// TIA Portal project "Project21" (V19)

(* hardware
DEVICE "S7-1200 station_1"  S7-1200 Station
   slot 0: "Rack_0"  S7-1200 Rack  Rack  V1.0
   slot 1: "PLC_1"  CPU 1215C DC/DC/DC  6ES7 215-1AG40-0XB0  V4.5
*)

// ===== PLC "PLC_1"  CPU 1215C DC/DC/DC =====

VAR_GLOBAL   // PLC tag table "Default tag table"
   "Encendido" AT %M0.0 : Bool;
   "ManAuto" AT %M0.1 : Bool;
   "System_Byte" AT %MB1 : Byte;
   "FirstScan" AT %M1.0 : Bool;
   "DiagStatusUpdate" AT %M1.1 : Bool;
   "AlwaysTRUE" AT %M1.2 : Bool;
   "AlwaysFALSE" AT %M1.3 : Bool;
END_VAR

DATA_BLOCK "DB_SimVent"   // DB1
{ S7_Optimized_Access := 'TRUE' }
VERSION : 0.1
// stored: InstanceOfName FB_Simulacion
"FB_Simulacion"
BEGIN
END_DATA_BLOCK

DATA_BLOCK "DB_HMIET"   // DB2
{ S7_Optimized_Access := 'FALSE' }
VERSION : 0.1
   VAR
      TEMPERATURA_SP : Real := 22.0;
      HUMEDAD_SP : Real := 60.0;
      PRESION_SP : Real := 1016.0;
      VENT_VEL_OUT : Real := 799.0;
      BOMBA_VEL_OUT : Real := 1434.0;
      CTRL_DESHUM : Int;
      CTRL_ENFRIAM_CALEF : Int;
      SPTEMP : Real;
      SPHUM : Real;
      SPPRE : Real;
      TEMPERATURA_HMI : Int;
      HUMEDAD_HMI : Int;
      PRESION_HMI : Int;
      ENFRIAMIENTO_HMI : Bool;
      CALEFACCION_HMI : Bool;
      DESHUM_HMI : Bool;
      AutoMan : Bool;
      SPTEMP_HMI : Real;
      SPHUM_HMI : Real;
      SPPRE_HMI : Real;
   END_VAR
BEGIN
END_DATA_BLOCK

DATA_BLOCK "DM_SimTemp"   // DB3
{ S7_Optimized_Access := 'TRUE' }
VERSION : 0.1
// stored: InstanceOfName FB_Simulacion
"FB_Simulacion"
BEGIN
   PVIn := 19.0;
END_DATA_BLOCK

DATA_BLOCK "DB_SimPresion"   // DB4
{ S7_Optimized_Access := 'TRUE' }
VERSION : 0.1
// stored: InstanceOfName FB_Simulacion
"FB_Simulacion"
BEGIN
   PVIn := 1000.0;
END_DATA_BLOCK

DATA_BLOCK "DB_SimHumedad"   // DB5
{ S7_Optimized_Access := 'TRUE' }
VERSION : 0.1
// stored: InstanceOfName FB_Simulacion
"FB_Simulacion"
BEGIN
   PVIn := 50.0;
END_DATA_BLOCK

DATA_BLOCK "DB_SimBomba"   // DB6
{ S7_Optimized_Access := 'TRUE' }
VERSION : 0.1
// stored: InstanceOfName FB_Simulacion
"FB_Simulacion"
BEGIN
END_DATA_BLOCK

DATA_BLOCK "DB_HMIOUT"   // DB7
{ S7_Optimized_Access := 'FALSE' }
VERSION : 0.1
   VAR
      PRESION_OUT : Real;
      HUMEDAD_OUT : Real;
      TEMPERATURA_OUT : Real;
   END_VAR
BEGIN
END_DATA_BLOCK

FUNCTION_BLOCK "FB_Simulacion"   // FB2, LAD
{ S7_Optimized_Access := 'TRUE' }
VERSION : 0.1
   VAR_INPUT
      Encendido : Bool;
      ManAuto : Bool;
      MS : Real;
      MI : Real;
      PVIn : Real;
      SP : Real;
   END_VAR
   VAR_OUTPUT
      PVOut : Real;
      Ctrl : Int;
   END_VAR
   VAR
      TON_Simulacion : TON_TIME;
      ResetTimerSim : Bool;
      Sim1 : Bool;
      Sim2 : Bool;
      Sim3 : Bool;
      Timer_Ajuste : TON_TIME;
      ResetTimerAjuste : Bool;
      Estado : Int;
      MSSP : Real;
      MISP : Real;
      FinSim1 : Bool;
      FinSim2 : Bool;
      EnclavEstado : Bool;
      Timer_ManAuto : TON_TIME;
   END_VAR
   VAR_TEMP   // added for the SCL form of the ladder/FBD networks
      _w1 : Bool;
      _w2 : Bool;
   END_VAR
BEGIN

REGION Network 1
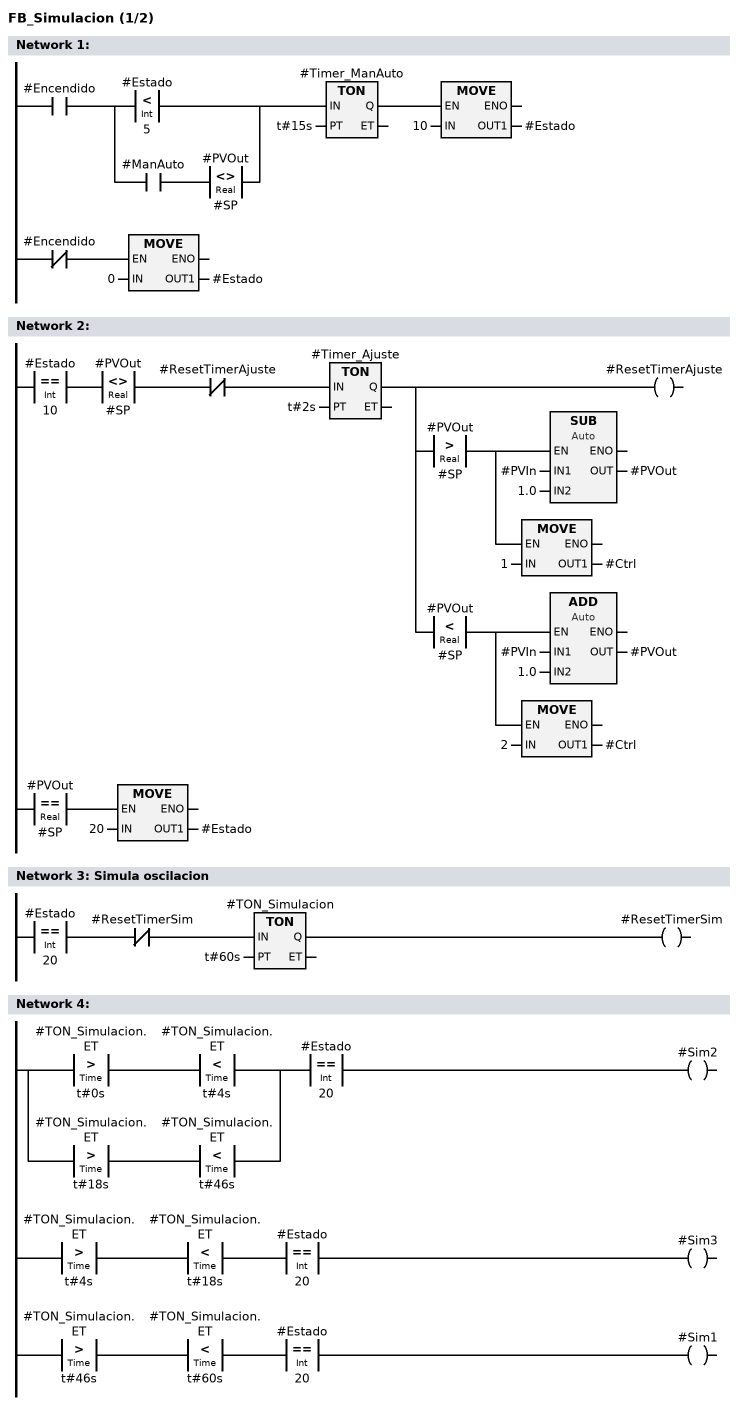
   #Timer_ManAuto(IN := #Encendido AND ((#Estado < 5) OR (#ManAuto AND (#PVOut <> #SP))), PT := t#15s);   // TON
   IF #Timer_ManAuto.Q THEN #Estado := 10; END_IF;
   IF NOT #Encendido THEN #Estado := 0; END_IF;
END_REGION

REGION Network 2
   #Timer_Ajuste(IN := (#Estado = 10) AND (#PVOut <> #SP) AND NOT #ResetTimerAjuste, PT := t#2s);   // TON
   #ResetTimerAjuste := #Timer_Ajuste.Q;
   #_w1 := #Timer_Ajuste.Q AND (#PVOut > #SP);
   IF #_w1 THEN
       #PVOut := #PVIn - 1.0;
       #Ctrl := 1;
   END_IF;
   #_w2 := #Timer_Ajuste.Q AND (#PVOut < #SP);
   IF #_w2 THEN
       #PVOut := #PVIn + 1.0;
       #Ctrl := 2;
   END_IF;
   IF #PVOut = #SP THEN #Estado := 20; END_IF;
END_REGION

REGION Network 3: Simula oscilacion
   #TON_Simulacion(IN := (#Estado = 20) AND NOT #ResetTimerSim, PT := t#60s);   // TON
   #ResetTimerSim := #TON_Simulacion.Q;
END_REGION

REGION Network 4
   RUNG wire#powerrail
      { S7_Templates := "SrcType := Time" } GT_Contact(in1 := #TON_Simulacion.ET, in2 := t#0s)
      { S7_Templates := "SrcType := Time" } LT_Contact(in1 := #TON_Simulacion.ET, in2 := t#4s)
      wire#w1
      { S7_Templates := "SrcType := Int" } EQ_Contact(in1 := #Estado, in2 := 20)
      Coil( #Sim2 )
   END_RUNG
   RUNG wire#powerrail
      { S7_Templates := "SrcType := Time" } GT_Contact(in1 := #TON_Simulacion.ET, in2 := t#18s)
      { S7_Templates := "SrcType := Time" } LT_Contact(in1 := #TON_Simulacion.ET, in2 := t#46s)
   END_RUNG wire#w1
   RUNG wire#powerrail
      { S7_Templates := "SrcType := Time" } GT_Contact(in1 := #TON_Simulacion.ET, in2 := t#4s)
      { S7_Templates := "SrcType := Time" } LT_Contact(in1 := #TON_Simulacion.ET, in2 := t#18s)
      { S7_Templates := "SrcType := Int" } EQ_Contact(in1 := #Estado, in2 := 20)
      Coil( #Sim3 )
   END_RUNG
   RUNG wire#powerrail
      { S7_Templates := "SrcType := Time" } GT_Contact(in1 := #TON_Simulacion.ET, in2 := t#46s)
      { S7_Templates := "SrcType := Time" } LT_Contact(in1 := #TON_Simulacion.ET, in2 := t#60s)
      { S7_Templates := "SrcType := Int" } EQ_Contact(in1 := #Estado, in2 := 20)
      Coil( #Sim1 )
   END_RUNG
   // the same network as SCL:
   #Sim2 := (((#TON_Simulacion.ET > t#0s) AND (#TON_Simulacion.ET < t#4s)) OR ((#TON_Simulacion.ET > t#18s) AND (#TON_Simulacion.ET < t#46s))) AND (#Estado = 20);
   #Sim3 := (#TON_Simulacion.ET > t#4s) AND (#TON_Simulacion.ET < t#18s) AND (#Estado = 20);
   #Sim1 := (#TON_Simulacion.ET > t#46s) AND (#TON_Simulacion.ET < t#60s) AND (#Estado = 20);
END_REGION

REGION Network 5
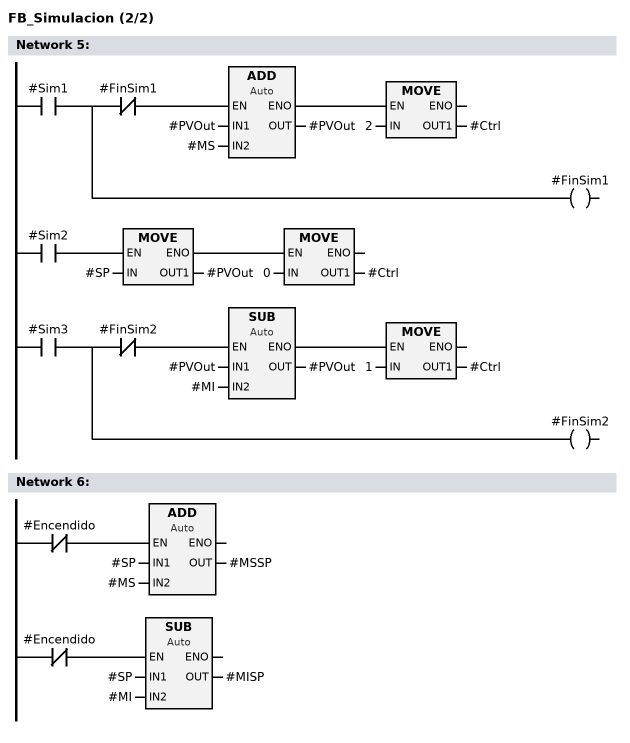
   RUNG wire#powerrail
      Contact( #Sim1 )
      wire#w1
      I_Contact( #FinSim1 )
      Add(in1 := #PVOut, in2 := #MS, out => #PVOut)
      Move(in := 2, out1 => #Ctrl)
   END_RUNG
   RUNG wire#w1
      Coil( #FinSim1 )
   END_RUNG
   RUNG wire#powerrail
      Contact( #Sim2 )
      Move(in := #SP, out1 => #PVOut)
      Move(in := 0, out1 => #Ctrl)
   END_RUNG
   RUNG wire#powerrail
      Contact( #Sim3 )
      wire#w2
      I_Contact( #FinSim2 )
      Sub(in1 := #PVOut, in2 := #MI, out => #PVOut)
      Move(in := 1, out1 => #Ctrl)
   END_RUNG
   RUNG wire#w2
      Coil( #FinSim2 )
   END_RUNG
   // the same network as SCL:
   IF #Sim1 AND NOT #FinSim1 THEN
       #PVOut := #PVOut + #MS;
       #Ctrl := 2;
   END_IF;
   #FinSim1 := #Sim1;
   IF #Sim2 THEN
       #PVOut := #SP;
       #Ctrl := 0;
   END_IF;
   IF #Sim3 AND NOT #FinSim2 THEN
       #PVOut := #PVOut - #MI;
       #Ctrl := 1;
   END_IF;
   #FinSim2 := #Sim3;
END_REGION

REGION Network 6
   RUNG wire#powerrail
      I_Contact( #Encendido )
      Add(in1 := #SP, in2 := #MS, out => #MSSP)
   END_RUNG
   RUNG wire#powerrail
      I_Contact( #Encendido )
      Sub(in1 := #SP, in2 := #MI, out => #MISP)
   END_RUNG
   // the same network as SCL:
   IF NOT #Encendido THEN
       #MSSP := #SP + #MS;
       #MISP := #SP - #MI;
   END_IF;
END_REGION
END_FUNCTION_BLOCK

FUNCTION "FC_ConversionEscalado" : Void   // FC1, LAD
{ S7_Optimized_Access := 'TRUE' }
VERSION : 0.1
   VAR_INPUT
      EntradaInt : Int;
      MinNorm : Int;
      MaxNorm : Int;
      MinReal : Real;
      MaxReal : Real;
   END_VAR
   VAR_OUTPUT
      SalidaReal : Real;
   END_VAR
   VAR_TEMP
      IntReal : Real;
      RealNorm : Real;
   END_VAR
BEGIN

REGION Network 1
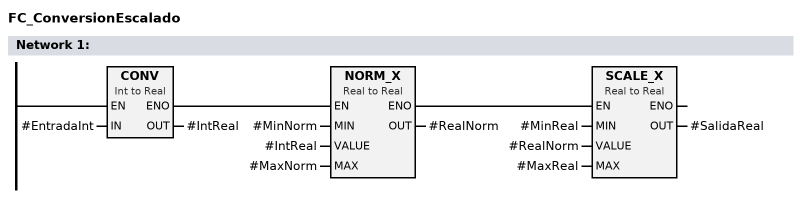
   RUNG wire#powerrail
      { S7_Templates := "[SrcType := Int, DestType := Real]" } Convert(in := #EntradaInt, out => #IntReal)
      { S7_Templates := "[SrcType := Real, DestType := Real]" } Normalize(min := #MinNorm, value := #IntReal, max := #MaxNorm, out => #RealNorm)
      { S7_Templates := "[SrcType := Real, DestType := Real]" } Scale(min := #MinReal, value := #RealNorm, max := #MaxReal, out => #SalidaReal)
   END_RUNG
   // the same network as SCL:
   #IntReal := INT_TO_REAL(#EntradaInt);
   #RealNorm := NORM_X(MIN := #MinNorm, VALUE := #IntReal, MAX := #MaxNorm);
   #SalidaReal := SCALE_X(MIN := #MinReal, VALUE := #RealNorm, MAX := #MaxReal);
END_REGION
END_FUNCTION

ORGANIZATION_BLOCK "Main"   // OB1, LAD, ProgramCycle
TITLE = "Main Program Sweep (Cycle)"
{ S7_Optimized_Access := 'TRUE' }
VERSION : 0.1
   VAR_INPUT
      Initial_Call : Bool;   // Initial call of this OB
      Remanence : Bool;   // =True, if remanent data are available
   END_VAR
   VAR_TEMP
      SPTEMP_ESC : Real;
      SPHUM_ESC : Real;
      SPPRE_ESC : Real;
   END_VAR
BEGIN

REGION Network 1
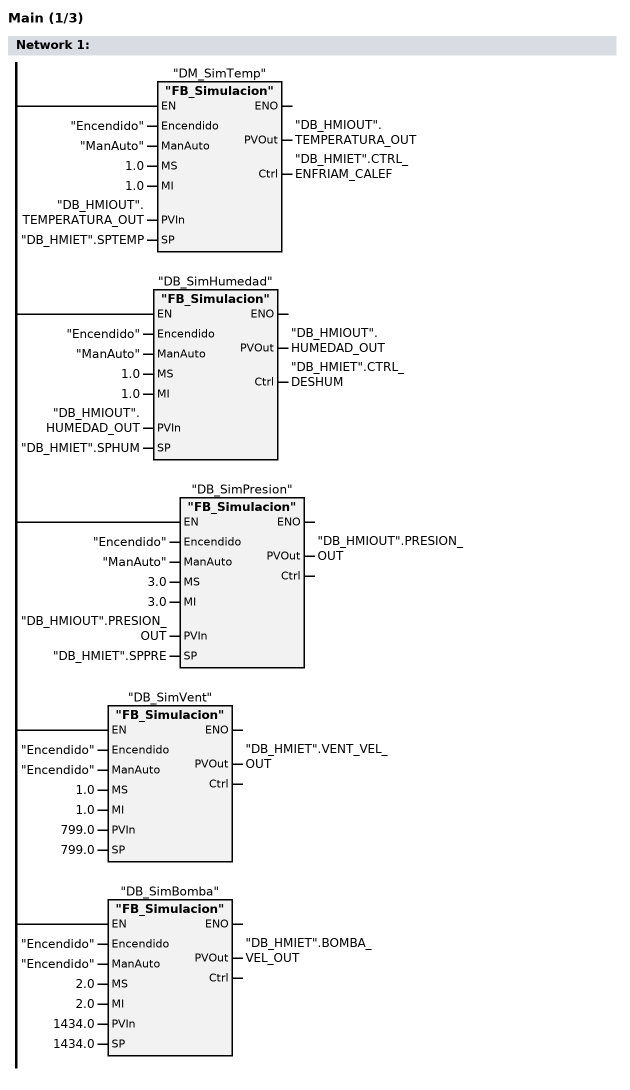
   RUNG wire#powerrail
      "DM_SimTemp"(Encendido := "Encendido", ManAuto := "ManAuto", MS := 1.0, MI := 1.0, PVIn := "DB_HMIOUT".TEMPERATURA_OUT, SP := "DB_HMIET".SPTEMP, PVOut => "DB_HMIOUT".TEMPERATURA_OUT, Ctrl => "DB_HMIET".CTRL_ENFRIAM_CALEF)
   END_RUNG
   RUNG wire#powerrail
      "DB_SimHumedad"(Encendido := "Encendido", ManAuto := "ManAuto", MS := 1.0, MI := 1.0, PVIn := "DB_HMIOUT".HUMEDAD_OUT, SP := "DB_HMIET".SPHUM, PVOut => "DB_HMIOUT".HUMEDAD_OUT, Ctrl => "DB_HMIET".CTRL_DESHUM)
   END_RUNG
   RUNG wire#powerrail
      "DB_SimPresion"(Encendido := "Encendido", ManAuto := "ManAuto", MS := 3.0, MI := 3.0, PVIn := "DB_HMIOUT".PRESION_OUT, SP := "DB_HMIET".SPPRE, PVOut => "DB_HMIOUT".PRESION_OUT, Ctrl =>)
   END_RUNG
   RUNG wire#powerrail
      "DB_SimVent"(Encendido := "Encendido", ManAuto := "Encendido", MS := 1.0, MI := 1.0, PVIn := 799.0, SP := 799.0, PVOut => "DB_HMIET".VENT_VEL_OUT, Ctrl =>)
   END_RUNG
   RUNG wire#powerrail
      "DB_SimBomba"(Encendido := "Encendido", ManAuto := "Encendido", MS := 2.0, MI := 2.0, PVIn := 1434.0, SP := 1434.0, PVOut => "DB_HMIET".BOMBA_VEL_OUT, Ctrl =>)
   END_RUNG
   // the same network as SCL:
   "DM_SimTemp"(Encendido := "Encendido",   // "FB_Simulacion"
                ManAuto := "ManAuto",
                MS := 1.0,
                MI := 1.0,
                PVIn := "DB_HMIOUT".TEMPERATURA_OUT,
                SP := "DB_HMIET".SPTEMP,
                PVOut => "DB_HMIOUT".TEMPERATURA_OUT,
                Ctrl => "DB_HMIET".CTRL_ENFRIAM_CALEF);
   "DB_SimHumedad"(Encendido := "Encendido",   // "FB_Simulacion"
                   ManAuto := "ManAuto",
                   MS := 1.0,
                   MI := 1.0,
                   PVIn := "DB_HMIOUT".HUMEDAD_OUT,
                   SP := "DB_HMIET".SPHUM,
                   PVOut => "DB_HMIOUT".HUMEDAD_OUT,
                   Ctrl => "DB_HMIET".CTRL_DESHUM);
   "DB_SimPresion"(Encendido := "Encendido",   // "FB_Simulacion"
                   ManAuto := "ManAuto",
                   MS := 3.0,
                   MI := 3.0,
                   PVIn := "DB_HMIOUT".PRESION_OUT,
                   SP := "DB_HMIET".SPPRE,
                   PVOut => "DB_HMIOUT".PRESION_OUT);
   "DB_SimVent"(Encendido := "Encendido",   // "FB_Simulacion"
                ManAuto := "Encendido",
                MS := 1.0,
                MI := 1.0,
                PVIn := 799.0,
                SP := 799.0,
                PVOut => "DB_HMIET".VENT_VEL_OUT);
   "DB_SimBomba"(Encendido := "Encendido",   // "FB_Simulacion"
                 ManAuto := "Encendido",
                 MS := 2.0,
                 MI := 2.0,
                 PVIn := 1434.0,
                 SP := 1434.0,
                 PVOut => "DB_HMIET".BOMBA_VEL_OUT);
END_REGION

REGION Network 2
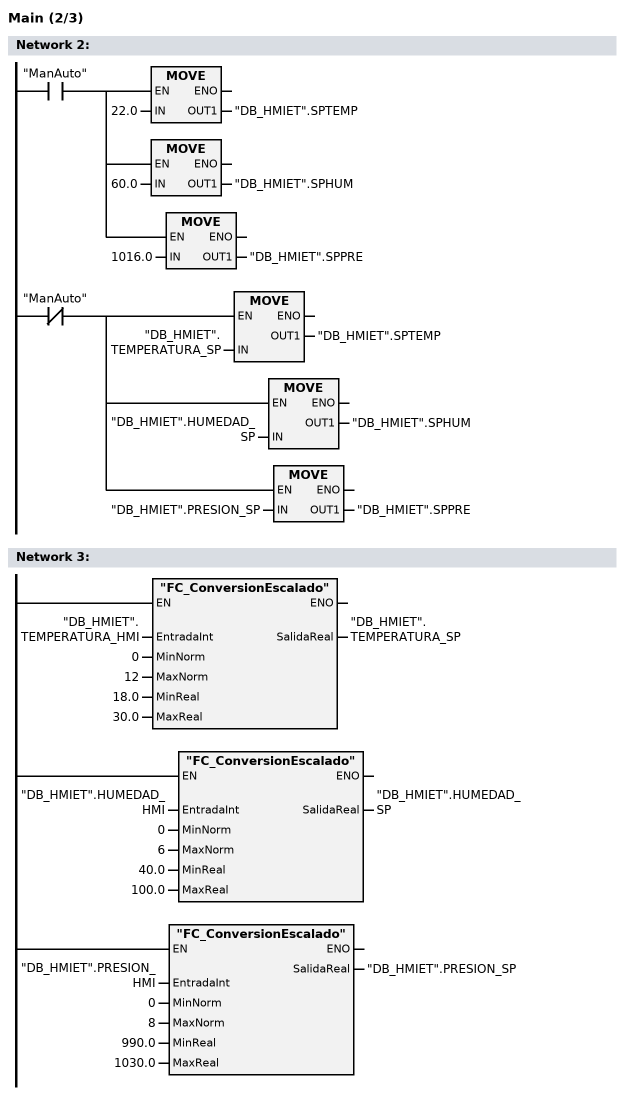
   RUNG wire#powerrail
      Contact( "ManAuto" )
      wire#w1
      Move(in := 22.0, out1 => "DB_HMIET".SPTEMP)
   END_RUNG
   RUNG wire#w1
      Move(in := 60.0, out1 => "DB_HMIET".SPHUM)
   END_RUNG
   RUNG wire#w1
      Move(in := 1016.0, out1 => "DB_HMIET".SPPRE)
   END_RUNG
   RUNG wire#powerrail
      I_Contact( "ManAuto" )
      wire#w2
      Move(in := "DB_HMIET".TEMPERATURA_SP, out1 => "DB_HMIET".SPTEMP)
   END_RUNG
   RUNG wire#w2
      Move(in := "DB_HMIET".HUMEDAD_SP, out1 => "DB_HMIET".SPHUM)
   END_RUNG
   RUNG wire#w2
      Move(in := "DB_HMIET".PRESION_SP, out1 => "DB_HMIET".SPPRE)
   END_RUNG
   // the same network as SCL:
   IF "ManAuto" THEN
       "DB_HMIET".SPTEMP := 22.0;
       "DB_HMIET".SPHUM := 60.0;
       "DB_HMIET".SPPRE := 1016.0;
   END_IF;
   IF NOT "ManAuto" THEN
       "DB_HMIET".SPTEMP := "DB_HMIET".TEMPERATURA_SP;
       "DB_HMIET".SPHUM := "DB_HMIET".HUMEDAD_SP;
       "DB_HMIET".SPPRE := "DB_HMIET".PRESION_SP;
   END_IF;
END_REGION

REGION Network 3
   RUNG wire#powerrail
      "FC_ConversionEscalado"(EntradaInt := "DB_HMIET".TEMPERATURA_HMI, MinNorm := 0, MaxNorm := 12, MinReal := 18.0, MaxReal := 30.0, SalidaReal => "DB_HMIET".TEMPERATURA_SP)
   END_RUNG
   RUNG wire#powerrail
      "FC_ConversionEscalado"(EntradaInt := "DB_HMIET".HUMEDAD_HMI, MinNorm := 0, MaxNorm := 6, MinReal := 40.0, MaxReal := 100.0, SalidaReal => "DB_HMIET".HUMEDAD_SP)
   END_RUNG
   RUNG wire#powerrail
      "FC_ConversionEscalado"(EntradaInt := "DB_HMIET".PRESION_HMI, MinNorm := 0, MaxNorm := 8, MinReal := 990.0, MaxReal := 1030.0, SalidaReal => "DB_HMIET".PRESION_SP)
   END_RUNG
   // the same network as SCL:
   "FC_ConversionEscalado"(EntradaInt := "DB_HMIET".TEMPERATURA_HMI,
                           MinNorm := 0,
                           MaxNorm := 12,
                           MinReal := 18.0,
                           MaxReal := 30.0,
                           SalidaReal => "DB_HMIET".TEMPERATURA_SP);
   "FC_ConversionEscalado"(EntradaInt := "DB_HMIET".HUMEDAD_HMI,
                           MinNorm := 0,
                           MaxNorm := 6,
                           MinReal := 40.0,
                           MaxReal := 100.0,
                           SalidaReal => "DB_HMIET".HUMEDAD_SP);
   "FC_ConversionEscalado"(EntradaInt := "DB_HMIET".PRESION_HMI,
                           MinNorm := 0,
                           MaxNorm := 8,
                           MinReal := 990.0,
                           MaxReal := 1030.0,
                           SalidaReal => "DB_HMIET".PRESION_SP);
END_REGION

REGION Network 4
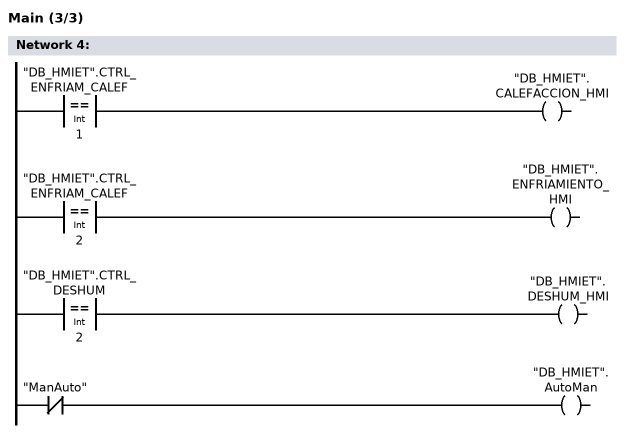
   RUNG wire#powerrail
      { S7_Templates := "SrcType := Int" } EQ_Contact(in1 := "DB_HMIET".CTRL_ENFRIAM_CALEF, in2 := 1)
      Coil( "DB_HMIET".CALEFACCION_HMI )
   END_RUNG
   RUNG wire#powerrail
      { S7_Templates := "SrcType := Int" } EQ_Contact(in1 := "DB_HMIET".CTRL_ENFRIAM_CALEF, in2 := 2)
      Coil( "DB_HMIET".ENFRIAMIENTO_HMI )
   END_RUNG
   RUNG wire#powerrail
      { S7_Templates := "SrcType := Int" } EQ_Contact(in1 := "DB_HMIET".CTRL_DESHUM, in2 := 2)
      Coil( "DB_HMIET".DESHUM_HMI )
   END_RUNG
   RUNG wire#powerrail
      I_Contact( "ManAuto" )
      Coil( "DB_HMIET".AutoMan )
   END_RUNG
   // the same network as SCL:
   "DB_HMIET".CALEFACCION_HMI := "DB_HMIET".CTRL_ENFRIAM_CALEF = 1;
   "DB_HMIET".ENFRIAMIENTO_HMI := "DB_HMIET".CTRL_ENFRIAM_CALEF = 2;
   "DB_HMIET".DESHUM_HMI := "DB_HMIET".CTRL_DESHUM = 2;
   "DB_HMIET".AutoMan := NOT "ManAuto";
END_REGION
END_ORGANIZATION_BLOCK